FUNCTION_BLOCK T_Counter
VAR
    Count : DINT;
END_VAR

METHOD Dec : DINT
VAR_INPUT
END_VAR
Count := Count - 1;
Dec := Count;
END_METHOD

METHOD Inc : DINT
VAR_INPUT
END_VAR
Count := Count + 1;
Inc := Count;
END_METHOD

METHOD Init
VAR_INPUT
	Value : DINT;
END_VAR
Count := Value;
END_METHOD

METHOD Reset
VAR_INPUT
END_VAR
Count := 0;
END_METHOD

PROPERTY Value : DINT
GET
Value := Count;
END_GET
END_PROPERTY

PROPERTY ValueAsTArg : T_Arg
GET
ValueAsTArg := F_DINT(Count);
END_GET
END_PROPERTY

END_FUNCTION_BLOCK

(* stored: Version 1.1.0.1, ProductVersion 3.1.4024.6
   POU T_Counter: Id {9ae51f40-0403-4a86-af5a-dd20e2f13d36}, SpecialFunc None
   Method Dec: Id {b171eb38-4d54-4cd6-ba87-90a20011def8}
   Method Inc: Id {5991a3e3-6db5-42ff-a03f-727af1168b75}
   Method Init: Id {871de783-64f5-4f07-ae83-1cbba81f7a2b}
   Method Reset: Id {cbcf06e0-d3ca-4315-8289-cb98c114d361}
   Property Value: Id {e951dec6-7422-4b6b-aa6c-19510cfee734}
   Get Get: Id {b2ac9b57-6bf7-42c8-a903-1b7f5f32981e}
   Property ValueAsTArg: Id {b4294afa-304a-49ee-9808-015ca4b4ff95}
   Get Get: Id {a9cee73b-b802-48ba-905a-a816c5c7cf4d} *)
